FUNCTION LetraPresente : BOOL
VAR_INPUT
	letra: STRING;
	cadena: STRING;
END_VAR
VAR
END_VAR

LetraPresente := FIND (cadena,letra) > 0;

END_FUNCTION

(* stored: Version 1.1.0.1, ProductVersion 3.1.4024.4
   POU LetraPresente: Id {50075678-603b-4616-8323-5471aeed9a5a}, SpecialFunc None *)
